{attribute 'qualified_only'}
VAR_GLOBAL
	Enc_Axis: AXIS_REF;
	Conveyor_Speed :	LREAL	;
	Encoder_Value	:	LREAL	;
	Real_Position: LREAL;
	Real_Velocity: LREAL;
	Count	AT%I*	:INT;
	Conveyor_CW AT%Q* : BOOL	;
	Conveyor_CCW AT%Q* : BOOL	;
	
END_VAR

(* stored: Version 1.1.0.1, ProductVersion 3.1.4024.15
   GVL GVL_Encoder: Id {5609fca6-061f-414c-859c-9bb76b705564} *)
